FUNCTION_BLOCK SS3_ifb_Axis (* Basic FB with empty ECC *)
  (* Standard: 61499-2 *)
  (* Version 1.0, 2021-08-23, AK121668 *)
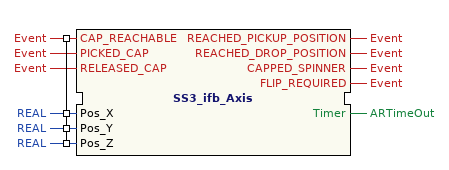
  EVENT_INPUT
    CAP_REACHABLE WITH Pos_X, Pos_Y, Pos_Z;
    PICKED_CAP;
    RELEASED_CAP;
  END_EVENT
  EVENT_OUTPUT
    REACHED_PICKUP_POSITION;
    REACHED_DROP_POSITION;
    CAPPED_SPINNER;
    FLIP_REQUIRED;
  END_EVENT
  VAR_INPUT
    Pos_X : REAL;
    Pos_Y : REAL;
    Pos_Z : REAL;
  END_VAR
  PLUGS
    Timer : ARTimeOut;
  END_PLUGS
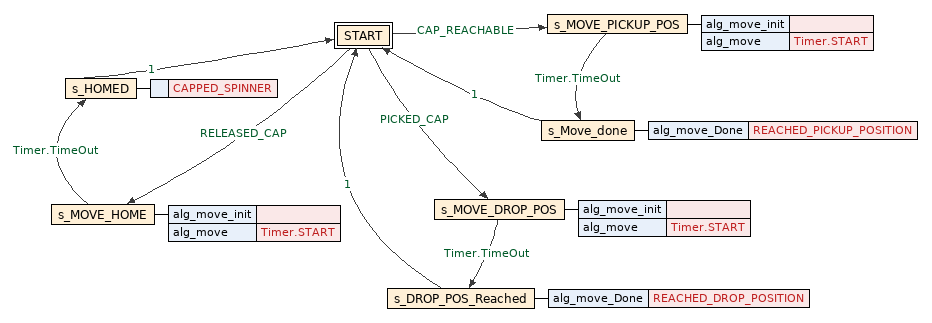
  EC_STATES
    START; (* Initial State *)
    s_MOVE_PICKUP_POS : alg_move_init, alg_move -> Timer.START;
    s_Move_done : alg_move_Done -> REACHED_PICKUP_POSITION;
    s_MOVE_DROP_POS : alg_move_init, alg_move -> Timer.START;
    s_DROP_POS_Reached : alg_move_Done -> REACHED_DROP_POSITION;
    s_MOVE_HOME : alg_move_init, alg_move -> Timer.START;
    s_HOMED : -> CAPPED_SPINNER;
  END_STATES
  EC_TRANSITIONS
    s_Move_done TO START := 1;
    START TO s_MOVE_PICKUP_POS := CAP_REACHABLE;
    s_MOVE_PICKUP_POS TO s_Move_done := Timer.TimeOut;
    s_DROP_POS_Reached TO START := 1;
    START TO s_MOVE_DROP_POS := PICKED_CAP;
    s_MOVE_DROP_POS TO s_DROP_POS_Reached := Timer.TimeOut;
    s_HOMED TO START := 1;
    START TO s_MOVE_HOME := RELEASED_CAP;
    s_MOVE_HOME TO s_HOMED := Timer.TimeOut;
  END_TRANSITIONS
  ALGORITHM alg_move_init IN ST:
Timer.DT := T#3s;
  END_ALGORITHM
  ALGORITHM alg_move IN ST:

  END_ALGORITHM
  ALGORITHM alg_move_Done IN ST:

  END_ALGORITHM
END_FUNCTION_BLOCK
